// TIA Portal project "SortingStation" (V15.1)
// Vorlageprojekt für das Buch mit Zielsystem S7-1200

(* hardware
DEVICE "S7-1200-Station_1"  S7-1200 Station
   slot 0: "Baugruppenträger_0"  Rack  V1.0
   slot 1: "PLC_1"  CPU 1211C DC/DC/DC  6ES7 211-1AE40-0XB0  V4.1
*)

// ===== PLC "PLC_1"  CPU 1211C DC/DC/DC =====

VAR_GLOBAL   // PLC tag table "Standard-Variablentabelle"
   "Entry Conveyor" AT %A0.0 : Bool;
   "At exit" AT %E0.0 : Bool;
   "Start" AT %E0.1 : Bool;
   "Stop" AT %I0.3 : Bool;
   "Exit Conveyor" AT %Q0.2 : Bool;
   "Sorter 1 belt" AT %Q0.4 : Bool;
   "Sorter 2 belt" AT %Q0.6 : Bool;
   "Sorter 3 belt" AT %Q1.0 : Bool;
   "Vision Sensor" AT %ID30 : DWord;
   "Sorter 2 turn" AT %Q0.5 : Bool;
   "Sorter 1 turn" AT %Q0.3 : Bool;
   "Sorter 3 turn" AT %Q0.7 : Bool;
   "DB_COND" AT %MD0 : DInt;
   "Reset" AT %I0.2 : Bool;
   "Counter 1" AT %QD30 : DWord;
   "Counter 2" AT %QD34 : DWord;
   "Counter 3" AT %QD38 : DWord;
END_VAR

// folder: System blocks/Program resources

DATA_BLOCK "Timer1"   // DB1
{ S7_Optimized_Access := 'TRUE' }
AUTHOR : Simatic
FAMILY : IEC
NAME : IEC_TMR
VERSION : 1.0
// stored: InstanceOfName IEC_TIMER
"IEC_TIMER"
BEGIN
END_DATA_BLOCK

DATA_BLOCK "Timer2"   // DB2
{ S7_Optimized_Access := 'TRUE' }
AUTHOR : Simatic
FAMILY : IEC
NAME : IEC_TMR
VERSION : 1.0
// stored: InstanceOfName IEC_TIMER
"IEC_TIMER"
BEGIN
END_DATA_BLOCK

DATA_BLOCK "Timer3"   // DB3
{ S7_Optimized_Access := 'TRUE' }
AUTHOR : Simatic
FAMILY : IEC
NAME : IEC_TMR
VERSION : 1.0
// stored: InstanceOfName IEC_TIMER
"IEC_TIMER"
BEGIN
END_DATA_BLOCK

DATA_BLOCK "Timer4"   // DB4
{ S7_Optimized_Access := 'TRUE' }
AUTHOR : Simatic
FAMILY : IEC
NAME : IEC_TMR
VERSION : 1.0
// stored: InstanceOfName IEC_TIMER
"IEC_TIMER"
BEGIN
END_DATA_BLOCK

DATA_BLOCK "Counter1"   // DB5
{ S7_Optimized_Access := 'TRUE' }
AUTHOR : Simatic
FAMILY : IEC
NAME : CNTR
VERSION : 1.0
// stored: InstanceOfName IEC_COUNTER
"IEC_COUNTER"
BEGIN
END_DATA_BLOCK

DATA_BLOCK "Counter2"   // DB6
{ S7_Optimized_Access := 'TRUE' }
AUTHOR : Simatic
FAMILY : IEC
NAME : CNTR
VERSION : 1.0
// stored: InstanceOfName IEC_COUNTER
"IEC_COUNTER"
BEGIN
END_DATA_BLOCK

DATA_BLOCK "Counter3"   // DB7
{ S7_Optimized_Access := 'TRUE' }
AUTHOR : Simatic
FAMILY : IEC
NAME : CNTR
VERSION : 1.0
// stored: InstanceOfName IEC_COUNTER
"IEC_COUNTER"
BEGIN
END_DATA_BLOCK

DATA_BLOCK "Timer5"   // DB8
{ S7_Optimized_Access := 'TRUE' }
AUTHOR : Simatic
FAMILY : IEC
NAME : IEC_TMR
VERSION : 1.0
// stored: InstanceOfName IEC_TIMER
"IEC_TIMER"
BEGIN
END_DATA_BLOCK

DATA_BLOCK "Timer6"   // DB9
{ S7_Optimized_Access := 'TRUE' }
AUTHOR : Simatic
FAMILY : IEC
NAME : IEC_TMR
VERSION : 1.0
// stored: InstanceOfName IEC_TIMER
"IEC_TIMER"
BEGIN
END_DATA_BLOCK

// folder: (top level)

FUNCTION "MHJ-PLC-Lab-Function-S71200" : Void   // FC9000, SCL
{ S7_Optimized_Access := 'TRUE' }
VERSION : 0.1
   VAR_TEMP
      rdTimeReturn : Int;
      outputTime : DTL;
      SyncVal : Byte;
      forVal : Int;
      forVal_2 : Int;
      Value : Byte;
   END_VAR
   VAR CONSTANT
      CompVal : Byte := 16#34;
      Value_01 : Byte := 16#11;
      Value_01_DW : DWord := 16#A165_D992;
      Value_02_DW : DWord := 16#58BE_4401;
   END_VAR
BEGIN

   #Value:=PEEK(area := 16#82,
        dbNumber := 0,
        byteOffset := 511);
   #Value := #Value + 1;

   POKE(area := 16#82,
        dbNumber := 0,
        byteOffset := 511,
        value := #Value);

   POKE(area:=16#81,
        dbNumber:=0,
        byteOffset:=1016,
        value:=#Value_01_DW);
   POKE(area := 16#81,
        dbNumber := 0,
        byteOffset := 1020,
        value := #Value_02_DW);

   POKE(area := 16#81,
        dbNumber := 0,
        byteOffset := 511,
        value := B#16#00);

   FOR #forVal := 0 TO 120 DO
       FOR #forVal_2:=0 TO 10 DO
           #rdTimeReturn:=RD_SYS_T(#outputTime);
           #rdTimeReturn := WR_SYS_T(#outputTime);
           #rdTimeReturn := RD_SYS_T(#outputTime);
           #rdTimeReturn := WR_SYS_T(#outputTime);
       END_FOR;
       #SyncVal:= PEEK(area := 16#81,
                      dbNumber := 0,
                      byteOffset := 511);
       IF #SyncVal = #CompVal THEN
          GOTO M_1;
       END_IF;
   END_FOR;
   RETURN;

   M_1:
   POKE(area := 16#81,
        dbNumber := 0,
        byteOffset := 511,
        value := B#16#0);
END_FUNCTION

ORGANIZATION_BLOCK "Main"   // OB1, LAD, ProgramCycle
TITLE = "Main Program Sweep (Cycle)"
{ S7_Optimized_Access := 'TRUE' }
VERSION : 0.1
   VAR_INPUT
      Initial_Call : Bool;   // Initial call of this OB
      Remanence : Bool;   // =True, if remanent data are available
   END_VAR
   VAR_TEMP   // added for the SCL form of the ladder/FBD networks
      _w1 : Bool;
      _w2 : Bool;
   END_VAR
BEGIN

REGION Network 1: Konnektierungsbaustein für PLC-Lab
   // Im Netzwerk 1 wird der Konnektierungsbaustein für PLC-Lab aufgerufen.
   // Dieser Aufruf darf nicht entfernt werden!
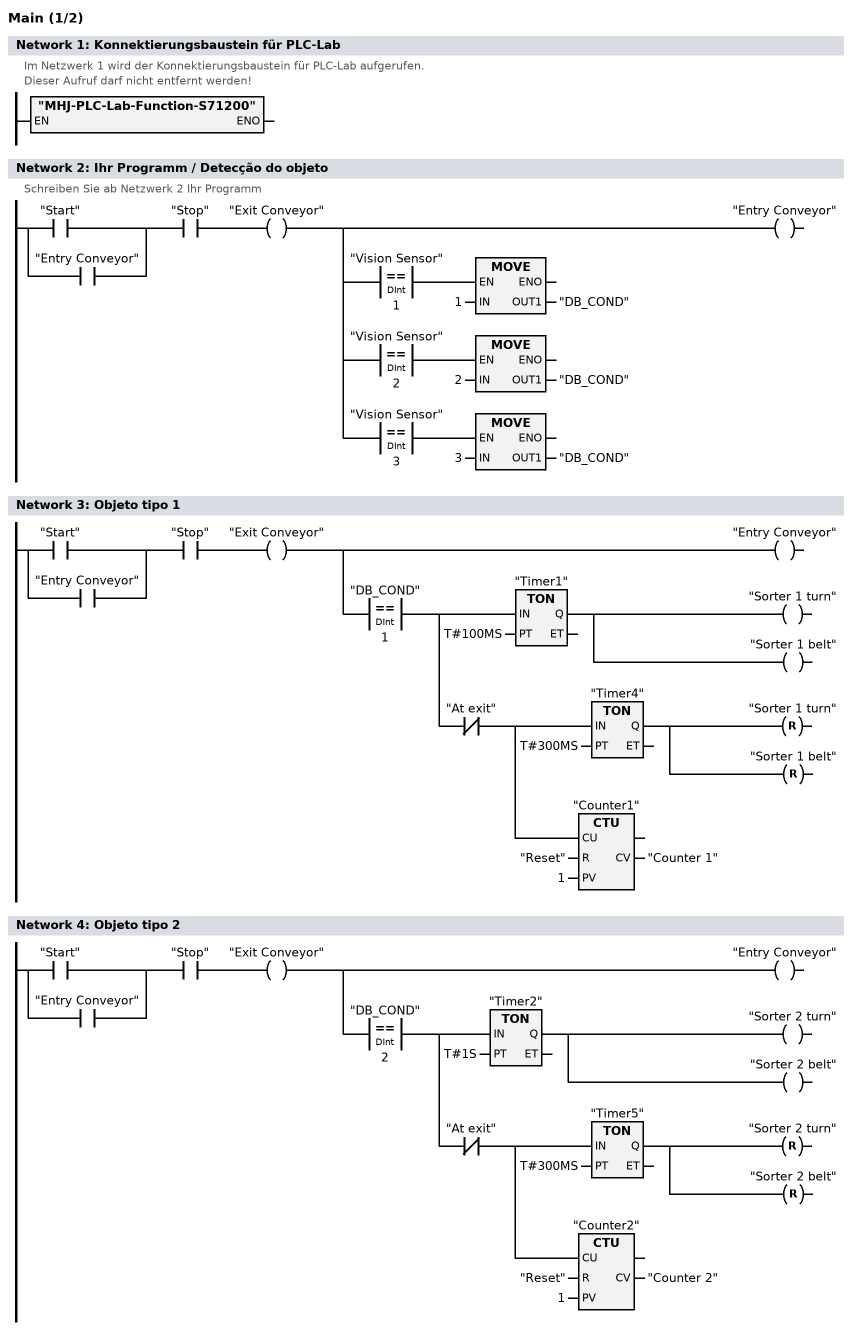
   RUNG wire#powerrail
      "MHJ-PLC-Lab-Function-S71200"()
   END_RUNG
   // the same network as SCL:
   "MHJ-PLC-Lab-Function-S71200"();
END_REGION

REGION Network 2: Ihr Programm / Detecção do objeto
   // Schreiben Sie ab Netzwerk 2 Ihr Programm
   RUNG wire#powerrail
      Contact( "Start" )
      wire#w1
      Contact( "Stop" )
      Coil( "Exit Conveyor" )
      wire#w2
      Coil( "Entry Conveyor" )
   END_RUNG
   RUNG wire#powerrail
      Contact( "Entry Conveyor" )
   END_RUNG wire#w1
   RUNG wire#w2
      { S7_Templates := "SrcType := DInt" } EQ_Contact(in1 := "Vision Sensor", in2 := 1)
      Move(in := 1, out1 => "DB_COND")
   END_RUNG
   RUNG wire#w2
      { S7_Templates := "SrcType := DInt" } EQ_Contact(in1 := "Vision Sensor", in2 := 2)
      Move(in := 2, out1 => "DB_COND")
   END_RUNG
   RUNG wire#w2
      { S7_Templates := "SrcType := DInt" } EQ_Contact(in1 := "Vision Sensor", in2 := 3)
      Move(in := 3, out1 => "DB_COND")
   END_RUNG
   // the same network as SCL:
   "Exit Conveyor" := ("Start" OR "Entry Conveyor") AND "Stop";
   "Entry Conveyor" := "Exit Conveyor";
   IF "Exit Conveyor" AND ("Vision Sensor" = 1) THEN "DB_COND" := 1; END_IF;
   IF "Exit Conveyor" AND ("Vision Sensor" = 2) THEN "DB_COND" := 2; END_IF;
   IF "Exit Conveyor" AND ("Vision Sensor" = 3) THEN "DB_COND" := 3; END_IF;
END_REGION

REGION Network 3: Objeto tipo 1
   "Exit Conveyor" := ("Start" OR "Entry Conveyor") AND "Stop";
   "Entry Conveyor" := "Exit Conveyor";
   #_w1 := "Exit Conveyor" AND ("DB_COND" = 1);
   "Timer1".TON(IN := #_w1, PT := T#100MS);
   "Sorter 1 turn" := "Timer1".Q;
   "Sorter 1 belt" := "Timer1".Q;
   #_w2 := #_w1 AND NOT "At exit";
   "Timer4".TON(IN := #_w2, PT := T#300MS);
   IF "Timer4".Q THEN
       "Sorter 1 turn" := FALSE;
       "Sorter 1 belt" := FALSE;
   END_IF;
   "Counter1".CTU(CU := #_w2, R := "Reset", PV := 1, CV => "Counter 1");
END_REGION

REGION Network 4: Objeto tipo 2
   "Exit Conveyor" := ("Start" OR "Entry Conveyor") AND "Stop";
   "Entry Conveyor" := "Exit Conveyor";
   #_w1 := "Exit Conveyor" AND ("DB_COND" = 2);
   "Timer2".TON(IN := #_w1, PT := T#1S);
   "Sorter 2 turn" := "Timer2".Q;
   "Sorter 2 belt" := "Timer2".Q;
   #_w2 := #_w1 AND NOT "At exit";
   "Timer5".TON(IN := #_w2, PT := T#300MS);
   IF "Timer5".Q THEN
       "Sorter 2 turn" := FALSE;
       "Sorter 2 belt" := FALSE;
   END_IF;
   "Counter2".CTU(CU := #_w2, R := "Reset", PV := 1, CV => "Counter 2");
END_REGION

REGION Network 5: Objeto tipo 3
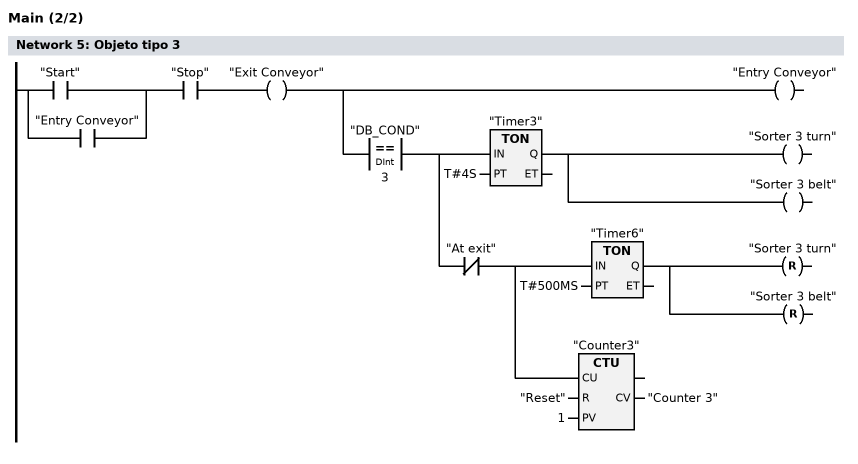
   "Exit Conveyor" := ("Start" OR "Entry Conveyor") AND "Stop";
   "Entry Conveyor" := "Exit Conveyor";
   #_w1 := "Exit Conveyor" AND ("DB_COND" = 3);
   "Timer3".TON(IN := #_w1, PT := T#4S);
   "Sorter 3 turn" := "Timer3".Q;
   "Sorter 3 belt" := "Timer3".Q;
   #_w2 := #_w1 AND NOT "At exit";
   "Timer6".TON(IN := #_w2, PT := T#500MS);
   IF "Timer6".Q THEN
       "Sorter 3 turn" := FALSE;
       "Sorter 3 belt" := FALSE;
   END_IF;
   "Counter3".CTU(CU := #_w2, R := "Reset", PV := 1, CV => "Counter 3");
END_REGION
END_ORGANIZATION_BLOCK